// TIA Portal V20 program export: 1 tag tables, 0 data types, 1 data blocks, 1 code blocks (in call order from the OBs), 0 instance data blocks

VAR_GLOBAL   // PLC tag table "Default tag table"
   on AT %M0.0 : Bool;
   off AT %M0.1 : Bool;
   lamp AT %Q8.0 : Bool;
   System_Byte AT %MB1 : Byte;
   FirstScan AT %M1.0 : Bool;
   DiagStatusUpdate AT %M1.1 : Bool;
   AlwaysTRUE AT %M1.2 : Bool;
   AlwaysFALSE AT %M1.3 : Bool;
   Clock_Byte AT %MB0 : Byte;
   Clock_10Hz AT %M0.0 : Bool;
   Clock_5Hz AT %M0.1 : Bool;
   "Clock_2.5Hz" AT %M0.2 : Bool;
   Clock_2Hz AT %M0.3 : Bool;
   "Clock_1.25Hz" AT %M0.4 : Bool;
   Clock_1Hz AT %M0.5 : Bool;
   "Clock_0.625Hz" AT %M0.6 : Bool;
   "Clock_0.5Hz" AT %M0.7 : Bool;
END_VAR

DATA_BLOCK "Data_block_1"   // DB1
TITLE = Motor
{ S7_Optimized_Access := 'TRUE' }
// stored: MemoryReserve 100
   VAR
      Motor_on : Bool := false;
      Motor_overload : Bool;
      Target_position : Int := 50;
   END_VAR
BEGIN
END_DATA_BLOCK

ORGANIZATION_BLOCK "Main"   // OB1, LAD, ProgramCycle
TITLE = "Main Program Sweep (Cycle)"
{ S7_Optimized_Access := 'TRUE' }
// stored: SetENOAutomatically false
   VAR_INPUT
      Initial_Call : Bool;   // Initial call of this OB
      Remanence : Bool;   // =True, if remanent data are available
   END_VAR
BEGIN

REGION Network 1
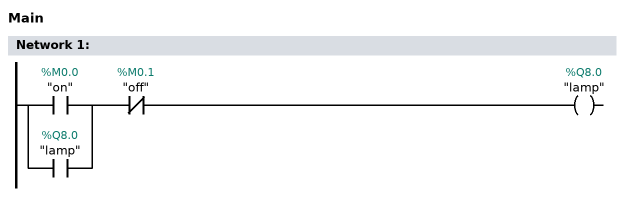
   RUNG wire#powerrail
      Contact( "on" )
      wire#w1
      I_Contact( "off" )
      Coil( "lamp" )
   END_RUNG
   RUNG wire#powerrail
      Contact( "lamp" )
   END_RUNG wire#w1
   // the same network as SCL:
   "lamp" := ("on" OR "lamp") AND NOT "off";
END_REGION
END_ORGANIZATION_BLOCK
